{attribute 'GeneratedUsingTerminal: EP3314-0002-0019'}
{attribute addProperty BoxType "EP3314-0002-0019"}
{attribute addProperty Id "TC_Inputs_Channel_1AT %I*AI_Standard_Channel_4A3944819TC_Inputs_Channel_2AT %I*AI_Standard_Channel_4A3944819TC_Inputs_Channel_3AT %I*AI_Standard_Channel_4A3944819TC_Inputs_Channel_4AT %I*AI_Standard_Channel_4A3944819WcStateAT %I*WcState_9091E0EB2InfoDataAT %I*InfoData_32EB74EA10"}
{attribute addProperty CRC "3864845084"}
{attribute addProperty Size "48"}
TYPE EP3314_E65CDB1C EXTENDS EtcSlaveBoxBase_77A0E4A7 :
STRUCT
	{attribute addProperty Name "TC_Inputs_Channel_1"}
	TC_Inputs_Channel_1 : AI_Standard_Channel_4A394481;
	{attribute addProperty Name "TC_Inputs_Channel_2"}
	TC_Inputs_Channel_2 : AI_Standard_Channel_4A394481;
	{attribute addProperty Name "TC_Inputs_Channel_3"}
	TC_Inputs_Channel_3 : AI_Standard_Channel_4A394481;
	{attribute addProperty Name "TC_Inputs_Channel_4"}
	TC_Inputs_Channel_4 : AI_Standard_Channel_4A394481;
	{attribute addProperty Name "WcState"}
	WcState : WcState_9091E0EB;
	{attribute addProperty Name "InfoData"}
	InfoData : InfoData_32EB74EA;
END_STRUCT
END_TYPE

(* stored: Version 1.2.0.0, ProductVersion 3.1.4024.9
   DUT EP3314_E65CDB1C: Id {26435d04-8411-4b6f-a362-007cd7329f92} *)
